FUNCTION_BLOCK FB_LightTower EXTENDS FB_Device
VAR_INPUT
	diStationState					: EN_StationStatus;
END_VAR
VAR
	Green	 			AT %Q* 		:BOOL;
	Ambar	 			AT %Q* 		:BOOL;
	Red		 			AT %Q* 		:BOOL;
	Buzzer 				AT %Q* 		:BOOL;
END_VAR

END_FUNCTION_BLOCK

(* stored: Version 1.1.0.1
   POU FB_LightTower: Id {f351574d-6f75-4144-ba3a-23a3745caf6f}, SpecialFunc None *)
